// TwinCAT 3 PLC project plc_kfe_vac
// ProgramVersion: 3.1.4022.4
// libraries:
//   LCLS General, * (SLAC)
//   LCLS Vacuum, * (SLAC - LCLS)
//   PMPS, * (SLAC - LCLS)
//   Tc2_Standard, * (Beckhoff Automation GmbH)
//   Tc2_System, * (Beckhoff Automation GmbH)
//   Tc2_Utilities, * (Beckhoff Automation GmbH)
//   Tc3_Module, * (Beckhoff Automation GmbH)
// project tree:
//   DUTs/ ST_EXT_ILK.TcDUT (not stored)
//   / FSV_task.TcTTO (not stored), PlcTask.TcTTO (not stored)
//   GVLs/ GVL_SXR_VAC.TcGVL (not stored), GVL_VAC_INTF.TcGVL (not stored), GVL_Variables.TcGVL (not stored), GVL_VFS.TcGVL (not stored)
//   POUs/ FB_AD_TREATY_GAUGE.TcPOU (not stored), FB_AD_TREATY_VGC.TcPOU (not stored), FB_EXT_ILK.TcPOU (not stored), MAIN.TcPOU (not stored), PRG_DIAGNOSTIC.TcPOU (not stored), PRG_PMPS.TcPOU (not stored), PRG_SXR_VAC.TcPOU, PRG_VAC_INTF.TcPOU (not stored), PRG_VFS.TcPOU (not stored)

// ---- POUs/PRG_SXR_VAC.TcPOU
PROGRAM PRG_SXR_VAC
VAR
END_VAR




// MKS275 Gauges

fb_MR1K1_BEND_GPI_1(PG=>);
fb_MR2K3_TXI_GPI_1(PG=>);
fb_MR1K3_TXI_GPI_1(PG=>);
fb_SP1K1_MONO_GPI_1(PG=>);
fb_TV3K0_GPI_1(PG=>);
fb_MR1K4_SOMS_GPI_1(PG=>);

// MKS500_EP Gauges

fb_MR1K1_BEND_GCC_1(PG := fb_MR1K1_BEND_GPI_1.PG, bEP:=TRUE);
fb_MR2K3_TXI_GCC_1(PG := fb_MR2K3_TXI_GPI_1.PG, bEP:=TRUE);
fb_MR1K3_TXI_GCC_1(PG := fb_MR1K3_TXI_GPI_1.PG, bEP:=TRUE);
fb_SP1K1_MONO_GCC_1(PG := fb_SP1K1_MONO_GPI_1.PG, bEP:=TRUE);
fb_TV3K0_GCC_1(PG := fb_TV3K0_GPI_1.PG, bEP:=TRUE);
fb_MR1K4_SOMS_GCC_1(PG := fb_MR1K4_SOMS_GPI_1.PG, bEP:=TRUE);

// VGC Valves

fb_RTDSK0_VGC_1( i_stUSG := fb_TV1K0_INTF_GCC_1.IG, i_stDSG := fb_RTDSK0_GCC_1.IG, i_xDis_DPIlk := FALSE,
                i_xEPS_OK := TRUE, i_xPMPS_OK := TRUE, i_xExt_OK := TRUE, i_xOverrideMode := xSystemOverrideMode,
                i_xReset := xReset_PMPS_FFO_K0, io_fbFFHWO := g_FastFaultOutputK0, fbArbiter := g_fbArbiter1 ,
                i_sDevName := 'RTDSK0:VGC:1' );

fb_EM1K0_GMD_VGC_1(i_stUSG := fb_RTDSK0_GCC_1.IG, i_stDSG := fb_EM1K0_GMD_GCC_10_reader.IG, i_xDis_DPIlk := FALSE,
                i_xEPS_OK := TRUE, i_xPMPS_OK := TRUE, i_xExt_OK := (NOT fb_EM1K0_GMD_GCC_10_reader.bError),
                   i_xOverrideMode := xSystemOverrideMode, i_xReset := xReset_PMPS_FFO_K0, io_fbFFHWO := g_FastFaultOutputK0,
                fbArbiter := g_fbArbiter1,  i_sDevName := 'EM1K0:GMD:VGC:1');

fb_AT1K0_GAS_VGC_1(i_stUSG := fb_SL1K0_PIP_1.q_IG, i_stDSG := fb_AT1K0_GAS_GCC_10_reader.IG, i_xDis_DPIlk := FALSE, i_xEPS_OK := TRUE, i_xPMPS_OK := TRUE,
                i_xExt_OK := (NOT fb_AT1K0_GAS_GCC_10_reader.bError), i_xOverrideMode := xSystemOverrideMode,
                i_xReset := xReset_PMPS_FFO_K0, io_fbFFHWO := g_FastFaultOutputK0, fbArbiter := g_fbArbiter1, i_sDevName := 'AT1K0:GAS:VGC:1' );

fb_EM2K0_XGMD_VGC_1(i_stUSG := fb_AT1K0_GAS_GCC_140_reader.IG, i_stDSG := fb_EM2K0_XGMD_GCC_10_reader.IG, i_xDis_DPIlk := FALSE, i_xEPS_OK := TRUE, i_xPMPS_OK := TRUE,
                i_xExt_OK := (NOT fb_AT1K0_GAS_GCC_140_reader.bError) AND (NOT fb_EM2K0_XGMD_GCC_10_reader.bError),
                i_xOverrideMode := xSystemOverrideMode, i_xReset := xReset_PMPS_FFO_K0, io_fbFFHWO := g_FastFaultOutputK0, fbArbiter := g_fbArbiter1, i_sDevName := 'EM2K0:XGMD:VGC:1');

fb_EM2K0_XGMD_VGC_2(i_stUSG := fb_EM2K0_XGMD_GCC_90_reader.IG, i_stDSG := fb_TV2K0_GCC_1.IG, i_xDis_DPIlk := FALSE, i_xEPS_OK := TRUE, i_xPMPS_OK := TRUE,
                i_xExt_OK := (NOT fb_EM2K0_XGMD_GCC_90_reader.bError), i_xOverrideMode := xSystemOverrideMode,
                i_xReset := xReset_PMPS_FFO_K0, io_fbFFHWO := g_FastFaultOutputK0, fbArbiter := g_fbArbiter1, i_sDevName := 'EM2K0:XGMD:VGC:2');

fb_TV2K0_VGC_1(i_stUSG := fb_TV2K0_GCC_1.IG, i_stDSG := fb_TV2K0_GCC_2.IG, i_xDis_DPIlk := FALSE, i_xEPS_OK := TRUE,
                 i_xPMPS_OK := TRUE, i_xExt_OK := fb_TV2K0_VFS_1_Interface.i_xVAC_FAULT_OK, i_xOverrideMode := xSystemOverrideMode, i_xReset := xReset_PMPS_FFO_K0,
                io_fbFFHWO := g_FastFaultOutputK0, fbArbiter := g_fbArbiter1, i_sDevName := 'TV2K0:VGC:1');

fb_MR1K1_BEND_VGC_1(i_stUSG :=  fb_PA1K0.q_IG, i_stDSG :=fb_MR1K1_BEND_PIP_1.q_IG, i_xDis_DPIlk := FALSE, i_xEPS_OK := TRUE, i_xPMPS_OK := TRUE,
                i_xExt_OK := fb_TV2K0_VFS_1_Interface.i_xVAC_FAULT_OK, i_xOverrideMode := xSystemOverrideMode, i_xReset := xReset_PMPS_FFO_K0,
                io_fbFFHWO := g_FastFaultOutputK0, fbArbiter := g_fbArbiter1,i_sDevName := 'MR1K1:BEND:VGC:1');

fb_MR1K3_TXI_VGC_1(i_stUSG := fb_MR1K1_BEND_PIP_1.q_IG, i_stDSG := fb_MR1K3_TXI_PIP_1.q_IG, i_xDis_DPIlk := FALSE, i_xEPS_OK := TRUE,
                i_xPMPS_OK := TRUE, i_xExt_OK := TRUE, i_xOverrideMode := xSystemOverrideMode, i_xReset := xReset_PMPS_FFO_K0,
                io_fbFFHWO := g_FastFaultOutputK0, fbArbiter := g_fbArbiter1, i_sDevName := 'MR1K3:TXI:VGC:1');

fb_SP1K1_MONO_VGC_1(i_stUSG := fb_MR2K3_TXI_PIP_1.q_IG, i_stDSG := fb_SP1K1_MONO_PIP_1.q_IG, i_xDis_DPIlk := FALSE,
                i_xEPS_OK := TRUE, i_xPMPS_OK := TRUE, i_xExt_OK := TRUE, i_xOverrideMode := xSystemOverrideMode,
                i_xReset := xReset_PMPS_FFO_K2, io_fbFFHWO := g_FastFaultOutputK2, fbArbiter := g_fbArbiter1, i_sDevName := 'SP1K1:MONO:VGC:1');

fb_SP1K1_MONO_VGC_2(i_stUSG := fb_SP1K1_MONO_PIP_1.q_IG, i_stDSG := fb_PC1K1_INTF_GCC_1.IG, i_xDis_DPIlk := FALSE,
                i_xEPS_OK := TRUE, i_xPMPS_OK := TRUE, i_xExt_OK := TRUE, i_xOverrideMode := xSystemOverrideMode,
                i_xReset := xReset_PMPS_FFO_K2, io_fbFFHWO := g_FastFaultOutputK2, fbArbiter := g_fbArbiter1, i_sDevName := 'SP1K1:MONO:VGC:2');

fb_IM1K3_PPM_VGC_1(i_stUSG := fb_MR2K3_TXI_PIP_1.q_IG, i_stDSG := fb_PC1K3_INTF_PIP_1.IG , i_xDis_DPIlk := FALSE, i_xEPS_OK := TRUE, i_xPMPS_OK := TRUE,
                i_xExt_OK := TRUE, i_xOverrideMode := xSystemOverrideMode, i_xReset := xReset_PMPS_FFO_K3, io_fbFFHWO := g_FastFaultOutputK3,
                fbArbiter := g_fbArbiter1, i_sDevName := 'IM1K3:PPM:VGC:1');

fb_TV3K0_VGC_1(i_stUSG := fb_MR2K3_TXI_PIP_1.q_IG, i_stDSG := fb_TV3K0_PIP_1.q_IG, i_xDis_DPIlk := FALSE, i_xEPS_OK := TRUE,
                i_xPMPS_OK := TRUE, i_xExt_OK := TRUE, i_xOverrideMode := xSystemOverrideMode, i_xReset := xReset_PMPS_FFO_K4,
                io_fbFFHWO := g_FastFaultOutputK4, fbArbiter := g_fbArbiter1, i_sDevName := 'TV3K0:VGC:1');

fb_MR1K4_SOMS_VGC_1(i_stUSG := fb_TV3K0_PIP_1.q_IG, i_stDSG := fb_MR1K4_SOMS_GCC_1.IG, i_xDis_DPIlk := FALSE, i_xEPS_OK := TRUE,
                i_xPMPS_OK := TRUE, i_xExt_OK := TRUE, i_xOverrideMode := xSystemOverrideMode, i_xReset := xReset_PMPS_FFO_K4, io_fbFFHWO := g_FastFaultOutputK4,
                fbArbiter := g_fbArbiter1, i_sDevName := 'MR1K4:SOMS:VGC:1');

fb_IM1K0_XTES_VGC_1(i_stUSG :=fb_IM1K0_XTES_GCC_1.IG , i_stDSG := fb_SL1K0_PIP_1.q_IG, i_xDis_DPIlk := FALSE, i_xEPS_OK := TRUE,
                i_xPMPS_OK := TRUE, i_xExt_OK := TRUE, i_xOverrideMode := xSystemOverrideMode, i_xReset := xReset_PMPS_FFO_K0,
                io_fbFFHWO := g_FastFaultOutputK0, fbArbiter := g_fbArbiter1, i_sDevName :='IM1K0:XTES:VGC:1');

// VFS Valves

fb_TV2K0_VFS_1_Interface(IG := fb_PCPM3B_GFS_1.IG);

// PIP_Gamma Pumps

fb_RTDSK0_PIP_1(	i_stGauge := fb_RTDSK0_GCC_1.IG,		i_xOverrideMode := xSystemOverrideMode);
fb_RTDSK0_PIP_2(	i_stGauge := fb_RTDSK0_GCC_1.IG,		i_xOverrideMode := xSystemOverrideMode);
fb_RTDSK0_PIP_3(	i_stGauge := fb_RTDSK0_GCC_1.IG,		i_xOverrideMode := xSystemOverrideMode);
fb_RTDSK0_PIP_4(	i_stGauge := fb_RTDSK0_GCC_1.IG,		i_xOverrideMode := xSystemOverrideMode);
fb_RTDSK0_PIP_5(	i_stGauge := fb_RTDSK0_GCC_1.IG,		i_xOverrideMode := xSystemOverrideMode);
fb_PCPM3B_PIP_1(	i_stGauge := fb_PCPM3B_GFS_1.IG,		i_xOverrideMode := xSystemOverrideMode);
fb_PA1K0_PIP_1(		i_stGauge := fb_PA1K0_GCC_1.IG,			i_xOverrideMode := xSystemOverrideMode);
fb_PA1K0(			i_stGauge := fb_PA1K0_GCC_1.IG,			i_xOverrideMode := xSystemOverrideMode);
fb_MR1K1_BEND_PIP_1(i_stGauge := fb_MR1K1_BEND_GPI_1.PG,	i_xOverrideMode := xSystemOverrideMode);
fb_MR1K3_TXI_PIP_1(	i_stGauge := fb_MR1K3_TXI_GCC_1.IG,		i_xOverrideMode := xSystemOverrideMode);
fb_MR2K3_TXI_PIP_1(	i_stGauge := fb_MR1K3_TXI_GCC_1.IG,		i_xOverrideMode := xSystemOverrideMode);
fb_SP1K1_MONO_PIP_1(i_stGauge := fb_SP1K1_MONO_GPI_1.PG,	i_xOverrideMode := xSystemOverrideMode);
fb_SP1K1_MONO_PIP_2(i_stGauge := fb_SP1K1_MONO_GPI_1.PG,	i_xOverrideMode := xSystemOverrideMode);
fb_TV3K0_PIP_1(		i_stGauge := fb_TV3K0_GCC_1.IG,			i_xOverrideMode := xSystemOverrideMode);
fb_SL1K0_PIP_1( 	i_stGauge := fb_SL1K0_POWER_GPI_1.PG,	i_xOverrideMode := xSystemOverrideMode); // New Ion Pump



// FB_MKS422

fb_RTDSK0_GCC_1(PG := fb_RTDSK0_GPI_1.PG);
fb_IM1K0_XTES_GCC_1(PG := fb_IM1K0_XTES_GPI_1.PG);
fb_PCPM3B_GFS_1(PG := fb_SL1K0_POWER_GPI_1.PG);
fb_SL1K0_POWER_GCC_1(PG := fb_SL1K0_POWER_GPI_1.PG);
fb_TV2K0_GCC_1(PG := fb_TV2K0_GPI_1.PG);
fb_TV2K0_GCC_2(PG := fb_TV2K0_GPI_2.PG);
fb_PA1K0_GCC_1(PG := fb_PA1K0_GPI_1.PG);

// FB_MKS317

fb_RTDSK0_GPI_1(PG=>);
fb_IM1K0_XTES_GPI_1(PG=>);
fb_SL1K0_POWER_GPI_1(PG=>);
fb_TV2K0_GPI_1(PG=>);
fb_TV2K0_GPI_2(PG=>);
fb_PA1K0_GPI_1(PG=>);

END_PROGRAM
